PROGRAM P_Outputs
VAR
	fbWinchValveOutput 			: FB_ValveOutput;
	fbDisplacementValveOutput 	: FB_DisplacementValveOutput;
	eStatus 					: E_Status; 
	bEnableWinch 				: BOOL;
	bEnableDisplacement 		: BOOL;
	bTest1 						: BOOL; 
	bTest2 						: BOOL;
	fbDisplacementControl	    : FB_DisplacementControl;
	fDisplacementControlSignal  : LREAL;
	fDisplacementNormalizedInput : LREAL := 1.0;
	bEndStopNegActive 			: BOOL;
	bEndStopPosActive 			: BOOL;
	//bEndStopOverride 			: BOOL; // THIS is at the HMI.bEndStopOverride now
	fWinchValveNormalizedInput  : LREAL;
	fWinchValveInput 			: LREAL;
	bMotionControlActive 		: BOOL;
	bEnableMotion 				: BOOL;
END_VAR

IF MAIN.eStatus = E_Status.Running THEN
	G_IO.bEnablePCDV := TRUE;
	G_IO.bWinchValveEnable := TRUE;
ELSE
	G_IO.bEnablePCDV := FALSE;	
	G_IO.bWinchValveEnable := FALSE;
END_IF

IF NOT(bMotionControlActive) THEN
	bEnableMotion := G_IO.bWinchEnable;
ELSIF bMotionControlActive AND 	P_MotionControl.bManualEnable THEN
	bEnableMotion := G_IO.bWinchEnable;
ELSIF bMotionControlActive AND 	P_MotionControl.bAutoEnable THEN
	bEnableMotion := P_MotionControl.bAutoEnable;	
ELSE
	bEnableMotion := FALSE;
END_IF

///////////////////// Winch //////////////////////////////
IF (MAIN.eStatus = E_Status.Running) AND bEnableMotion THEN 
	G_IO.bOpenBrakes := TRUE;
	bEnableWinch := TRUE;
ELSE
	G_IO.bOpenBrakes := FALSE;
	bEnableWinch := FALSE;
END_IF


	

///////////////////// Displacement //////////////////////////////
IF (MAIN.eStatus = E_Status.Running) AND G_IO.bDisplacementEnable THEN 
	bEnableDisplacement := TRUE;
ELSE
	bEnableDisplacement := FALSE;
END_IF

IF NOT(bMotionControlActive) THEN
	fWinchValveInput := G_Sensors.fJoystickNormalizedY;
ELSE
	fWinchValveInput := P_MotionControl.fWinchControlOutput;
END_IF

IF P_MotionControl.fWinchPos < G_Parameters.stParam.fWinchEndStopNeg  AND NOT(HMI.bEndStopOverride) THEN
	bEndStopPosActive := FALSE;
	bEndStopNegActive := TRUE;
	fWinchValveNormalizedInput := LIMIT(-1.0, fWinchValveInput, 0.0);
ELSIF P_MotionControl.fWinchPos > G_Parameters.stParam.fWinchEndStopPos AND NOT(HMI.bEndStopOverride) THEN
	bEndStopPosActive := TRUE;
	bEndStopNegActive := FALSE;
	fWinchValveNormalizedInput := LIMIT(0, fWinchValveInput, 1.0);
ELSE
	bEndStopPosActive := FALSE;
	bEndStopNegActive := FALSE;
	fWinchValveNormalizedInput := fWinchValveInput;
END_IF



fbWinchValveOutput(
	bEnable := bEnableWinch,
	bDeadBandCompOn := G_Parameters.stParam.bWinchDeadBandCompOn,
	stValveDeadBand := G_Parameters.stParam.stWinchValveDeadBand,
	fNormalizedInput := fWinchValveNormalizedInput,
	bEnableValveOutput => bTest1,
	nOutput => G_IO.fWinchValveOut
);

//fbDisplacementControl(
//	bEnable := (MAIN.eStatus = E_Status.Running) AND NOT(bEnableDisplacement),
//	fProportionalGain := G_Parameters.stParam.fDisplacementControlPgain,
//	fDisplacementNormalizedInput :=  LIMIT(0.1, fDisplacementNormalizedInput, 1.0),
//	fYokeNormalizedFeedback := G_Sensors.fYokeNormalizedFeedback
//);

//// Dplacemot of the motor //////

IF NOT(bEnableDisplacement) THEN
	fDisplacementControlSignal := P_MotionControl.fDisplacementControlSignal; 
ELSE	
	fDisplacementControlSignal := G_Sensors.fJoystickNormalizedZ;
END_IF

fbDisplacementValveOutput(
	bEnable := (MAIN.eStatus = E_Status.Running) ,
	bDeadBandCompOn := G_Parameters.stParam.bDisplacementDeadBandCompOn,
	stValveDeadBand := G_Parameters.stParam.stDisplacementValveDeadBand,
	fNormalizedInput := fDisplacementControlSignal,
	bEnableValveOutput => bTest2,
	nOutput => G_IO.fWinchPDCVOut
);







///////// Swich form Manuel to Motion Control /////
IF (HMI.bStartTB) THEN 
	bMotionControlActive := TRUE; 
ELSE 
	bMotionControlActive  := FALSE; 	
END_IF

END_PROGRAM

(* stored: Version 1.1.0.1, ProductVersion 3.1.4024.12
   POU P_Outputs: Id {05725e2c-789e-4faf-9ddc-3f7ec72a2093}, SpecialFunc None *)
